{attribute 'qualified_only'}
VAR_GLOBAL CONSTANT
	// Encoder reference values in counts = nm
	nM1K1bendUS_ENC_REF : ULINT := 13376858;
	nM1K1bendDS_ENC_REF : ULINT := 14336722;
END_VAR

(* stored: Version 1.1.0.1, ProductVersion 3.1.4022.18
   GVL GVL_M1K1_Constants: Id {0f41f14c-3122-4f9d-824a-be5d7042bc4c} *)
